{attribute addProperty BoxType "EP9224-0023-0016"}
{attribute addProperty Id "DPO_Inputs_ChannelAT %I*ARRAY[0..39] OF DPO_Inputs_Channel_3CD9BEA3480600DPO_Inputs_DeviceAT %I*DPO_Inputs_Device_301DB633176220DPO_Outputs_ChannelAT %Q*ARRAY[0..12] OF DPO_Outputs_Channel_5760563F128160DPO_Outputs_DeviceAT %Q*DPO_Outputs_Device_6EB864581620WcStateAT %I*WcState_98A4DF7520.250InfoDataAT %I*InfoData_BC63D37F80100"}
{attribute addProperty CRC "902323771"}
{attribute addProperty SizeInBites "882"}
{attribute addProperty SizeInBytes "110.25"}
TYPE EP9224_D133F73C :
STRUCT
	{attribute addProperty Name "DPO_Inputs_Channel"}
	DPO_Inputs_Channel : ARRAY[0..39] OF DPO_Inputs_Channel_3CD9BEA3;
	{attribute addProperty Name "DPO_Inputs_Device"}
	DPO_Inputs_Device : DPO_Inputs_Device_301DB633;
	{attribute addProperty Name "DPO_Outputs_Channel"}
	DPO_Outputs_Channel : ARRAY[0..12] OF DPO_Outputs_Channel_5760563F;
	{attribute addProperty Name "DPO_Outputs_Device"}
	DPO_Outputs_Device : DPO_Outputs_Device_6EB86458;
	{attribute addProperty Name "WcState"}
	WcState : WcState_98A4DF75;
	{attribute addProperty Name "InfoData"}
	InfoData : InfoData_BC63D37F;
END_STRUCT
END_TYPE

(* stored: Version 1.2.0.0, ProductVersion 3.1.4024.9
   DUT EP9224_D133F73C: Id {a62dabea-ffaa-4306-a1f5-19d29578ed7d} *)
